(*********************************** G.D S.p.A. - Technical Department ***********************************
============= PROGRAM INFO ============
FOLDER:             TBD
MACHINES INVOLVED:  TBD 

============= DESCRIPTION =============
csp machine declaration

============= REVISIONS ===============
Date		Version	 	Author      	Description             
----------	-------		------------  	--------------------------------------------
2019/04/05 	0000.00	 	M.Grasso		Creation of the PRG

**********************************************************************************************************)
(*$R process_ref := prc; $*)
PROGRAM csp_case_transport_accU
VAR
	
	prc:											process;
	prc_path:										STRING;
	
END_VAR

_read_var_input();

_object_manager();

IF NOT objects_running()
THEN
	RETURN;	
END_IF

_read_process_image();

_mode_manager();
CASE process_get_mode(prc) OF
	MODE_ABSENT,
	MODE_INACTIVE:
		RETURN;
	MODE_TEST:
		_handle_process_test();
END_CASE
_set_runtime_properties();

(********************************* BODY *********************************)
(************************************************************************)

_handle_messages();

_write_output();

ACTION _handle_messages:
;
END_ACTION

ACTION _handle_process_test:
;
END_ACTION

ACTION _mode_manager:
IF process_mode_req_is_pending(prc)
THEN
    process_apply_mode_req_first_step(prc);
    CASE process_get_mode(prc) OF
        MODE_TO_ABSENT:
			;
        MODE_TO_INACTIVE:
			;
        MODE_TO_TEST:
			;
        MODE_TO_OPERATIONAL:
			;
    END_CASE
    process_apply_mode_req_second_step(prc);
END_IF
END_ACTION

ACTION _object_manager:
IF objects_initialization()
THEN
	sub_process_init(
		object_name					:= 'csp_case_transport_accU.prc', 
		process						:= csp_case_transport.prc, 
		CONVERSION_this				:= prc);
		
	prc_path 						:= process_get_path(prc);
END_IF

IF objects_running()
THEN
	process_cycle(prc);
END_IF
END_ACTION

ACTION _read_process_image:
;
END_ACTION

ACTION _read_var_input:
;
END_ACTION

ACTION _set_runtime_properties:
;
END_ACTION

ACTION _write_output:
;
END_ACTION

END_PROGRAM

(* stored: Version 1.1.0.1, ProductVersion 3.1.4024.3
   POU csp_case_transport_accU: Id {5c6a12e2-22f5-46e9-99f8-9b99fbeb8246}, SpecialFunc None
   Action _handle_messages: Id {3588cbb9-517f-4e66-9058-916568bed821}
   Action _handle_process_test: Id {33e02b88-459c-4398-ae8b-36ac0f298c81}
   Action _mode_manager: Id {45a39c3e-454a-43c0-9e92-5c1d6b7d28ec}
   Action _object_manager: Id {355cf21a-d666-4326-a6df-677ac8e33881}
   Action _read_process_image: Id {2e70abc5-3164-40bb-8632-4357a78f7992}
   Action _read_var_input: Id {a942a730-8578-4e4d-b24b-b6c5fddc4ced}
   Action _set_runtime_properties: Id {57c234e6-8afc-405c-bff4-bfab00b7dfe6}
   Action _write_output: Id {9964d143-12c0-4e33-867d-d0a510842e9f} *)
